{attribute 'qualified_only'}
{attribute 'strict'}
TYPE eProcessSequence :
(
	ComponentReady:=1,
	WaitingOpenGripper:=2,
	WaitingCloseGripper:=3,
	Busy := 254,
	Done :=255
);
END_TYPE

(* stored: Version 1.1.0.1, ProductVersion 3.1.4024.12
   DUT eProcessSequence: Id {b236de43-2b4c-0da2-0890-b808ca5b0db3} *)
